Yaskawa INFORM job: R2_W37-38-A1(90,180)_MP_OK.JBI

/JOB
//NAME R2_W37-38-A1(90,180)_MP_OK
///FOLDERNAME MP_TEST
//POS
///NPOS 26,26,0,2,0,0
///TOOL 0
///POSTYPE PULSE
///PULSE
C00000=93749,-89371,-91277,8096,41280,-46437
C00001=108253,34882,1520,-5365,47806,-39628
C00002=107169,33741,260,-4415,47933,-40104
C00003=108304,35007,6119,-5659,45057,-39444
C00004=108304,34897,6936,-5716,44500,-39408
C00005=97032,44199,11533,25896,52196,-55743
C00006=92155,59959,24555,42711,72963,-63593
C00007=93253,58543,22950,42257,72649,-63232
C00008=105844,23507,-13733,18910,63558,-49167
C00009=107323,34805,4423,-4698,45932,-39936
C00010=107323,34805,4423,-4698,45932,-39936
C00011=107323,34805,4423,-4698,45932,-39936
C00012=107323,34936,3725,-4660,46427,-39962
C00013=107323,35319,2035,-4568,47660,-40022
C00014=107312,34619,4228,39648,53886,-78090
C00015=110358,28426,690,32214,48246,-74412
C00016=107521,33383,7983,33979,44457,-77823
C00017=106695,32839,6145,41016,52545,-79043
C00018=107308,34320,6388,40349,52737,-78625
C00019=107316,34145,8806,34203,44441,-77946
C00020=107311,34069,8817,34225,44407,-77965
C00021=107311,34116,8051,33947,44823,-77787
C00022=107310,34362,5652,33086,46171,-77232
C00023=106870,9616,-25198,30572,51697,-75428
C00024=101735,-85908,-75899,60499,32479,-90887
C00025=45194,-87749,-78830,51897,50435,-40322
BC00000=142986,236852,53
BC00001=142986,236852,53
BC00002=141179,228534,53
BC00003=141179,228534,53
BC00004=141179,228534,53
BC00005=141038,227723,53
BC00006=152460,220216,3191
BC00007=152460,220216,3191
BC00008=173099,205796,53
BC00009=137305,226012,53
BC00010=137299,223707,53
BC00011=137305,226012,53
BC00012=137862,228620,53
BC00013=139253,235140,53
BC00014=200586,225503,53
BC00015=196056,221511,53
BC00016=180368,227117,53
BC00017=194244,219914,53
BC00018=194244,219914,53
BC00019=180368,227117,53
BC00020=204304,206217,53
BC00021=205743,208135,53
BC00022=209341,212930,53
BC00023=209341,212930,53
BC00024=209341,212930,53
BC00025=209341,212930,53
///POSTYPE BASE
///RECTAN
///RCONF 0,0,0,0,1,0,0,0,0,0,0,0,0,0,0,0,0,0,0,0,0,0,0,0
P00006=2.006,1.622,-0.565,0.0000,0.0000,0.0000
///RCONF 0,0,0,0,0,0,0,0,0,0,0,0,0,0,0,0,0,0,0,0,0,0,0,0
P00023=-2.957,-4.083,2.762,0.0000,0.0000,0.0000
//INST
///DATE 2023/11/16 10:53
///ATTR SC,RW
///GROUP1 RB1,BS1
NOP
'r2_W37-38-A1(90,180)
'
'Path S951
SFTOF
MOVJ C00000 BC00000 VJ=20.00
MOVL C00001 BC00001 V=100.0
MOVL C00002 BC00002 V=100.0
MOVL C00003 BC00003 V=60.0
REFP 3 C00004 BC00004
CALL JOB:SEARCH-R1
SET P023 P006
SFTON P023
MOVL C00005 BC00005 V=60.0
MOVL C00006 BC00006 V=60.0
REFP 3 C00007 BC00007
CALL JOB:SEARCH-R1
SET P023 P006
SFTON P023
MOVL C00008 BC00008 V=60.0
MOVL C00009 BC00009 V=60.0
REFP 3 C00010 BC00010
CALL JOB:SEARCH-R1
SET P023 P006
SFTON P023
MOVL C00011 BC00011 V=60.0
MOVL C00012 BC00012 V=100.0
MOVL C00013 BC00013 V=100.0
'Path W952
SFTOF
SFTON P023
MOVJ C00014 BC00014 VJ=20.00
MOVL C00015 BC00015 V=100.0
MACRO1 MJ#(0) ARGF8
MOVL C00016 BC00016 V=100.0 PL=0
REFP 1 C00017 BC00017
REFP 2 C00018 BC00018
ARCON
MOVL C00019 BC00019 V=10.0
MOVL C00020 BC00020 V=10.0
ARCOF
MOVL C00021 BC00021 V=100.0
MOVL C00022 BC00022 V=100.0
SFTOF
MOVJ C00023 BC00023 VJ=20.00
MOVJ C00024 BC00024 VJ=20.00
MOVJ C00025 BC00025 VJ=20.00
END
